// TIA Portal V19 export
TYPE "C106_VAR_REL_TYPIC"
   STRUCT
      AUT_STS { ExternalAccessible := 'False'; ExternalVisible := 'False'; ExternalWritable := 'False'} : USInt;   // Status van de vermogenschakelaar van de hoogspanning
   END_STRUCT;
END_TYPE
